REGION Network 13: CALL FB31 SPINDLE C24
   // 2#0000_0001 OPTIONS 0 BIT 0 MEASURING SYSTEM 2 OPTION
   // 2#0000_0010 OPTIONS 0 BIT 1 BELT BROKEN OPTION
   // 2#0000_0100 OPTIONS 0 BIT 2 COOLING OPTION
   // 2#0000_1000 OPTIONS 0 BIT 3 MQL OR HP OPTION
   // 2#0001_0000 OPTIONS 0 BIT 4 ANALOG TEMPERATURE SENSOR OPTION
   // 2#0010_0000 OPTIONS 0 BIT 5 PTC TEMPERATURE SENSOR OPTION
   // 2#0100_0000 OPTIONS 0 BIT 6 TWIN KESSLER VPM READY OPTION
   // 2#1000_0000 OPTIONS 0 BIT 7 MPP SPINDLE OVERRIDE OPTION
   // 
   // 2#0000_0001 OPTIONS 1 BIT 0 SPARE OPTION
   // 2#0000_0010 OPTIONS 1 BIT 1 SPARE OPTION
   // 2#0000_0100 OPTIONS 1 BIT 2 SPARE OPTION
   // 2#0000_1000 OPTIONS 1 BIT 3 SPARE OPTION
   // 2#0001_0000 OPTIONS 1 BIT 4 SPARE OPTION
   // 2#0010_0000 OPTIONS 1 BIT 5 SPARE OPTION
   // 2#0100_0000 OPTIONS 1 BIT 6 SPARE OPTION
   // 2#1000_0000 OPTIONS 1 BIT 7 SPARE OPTION
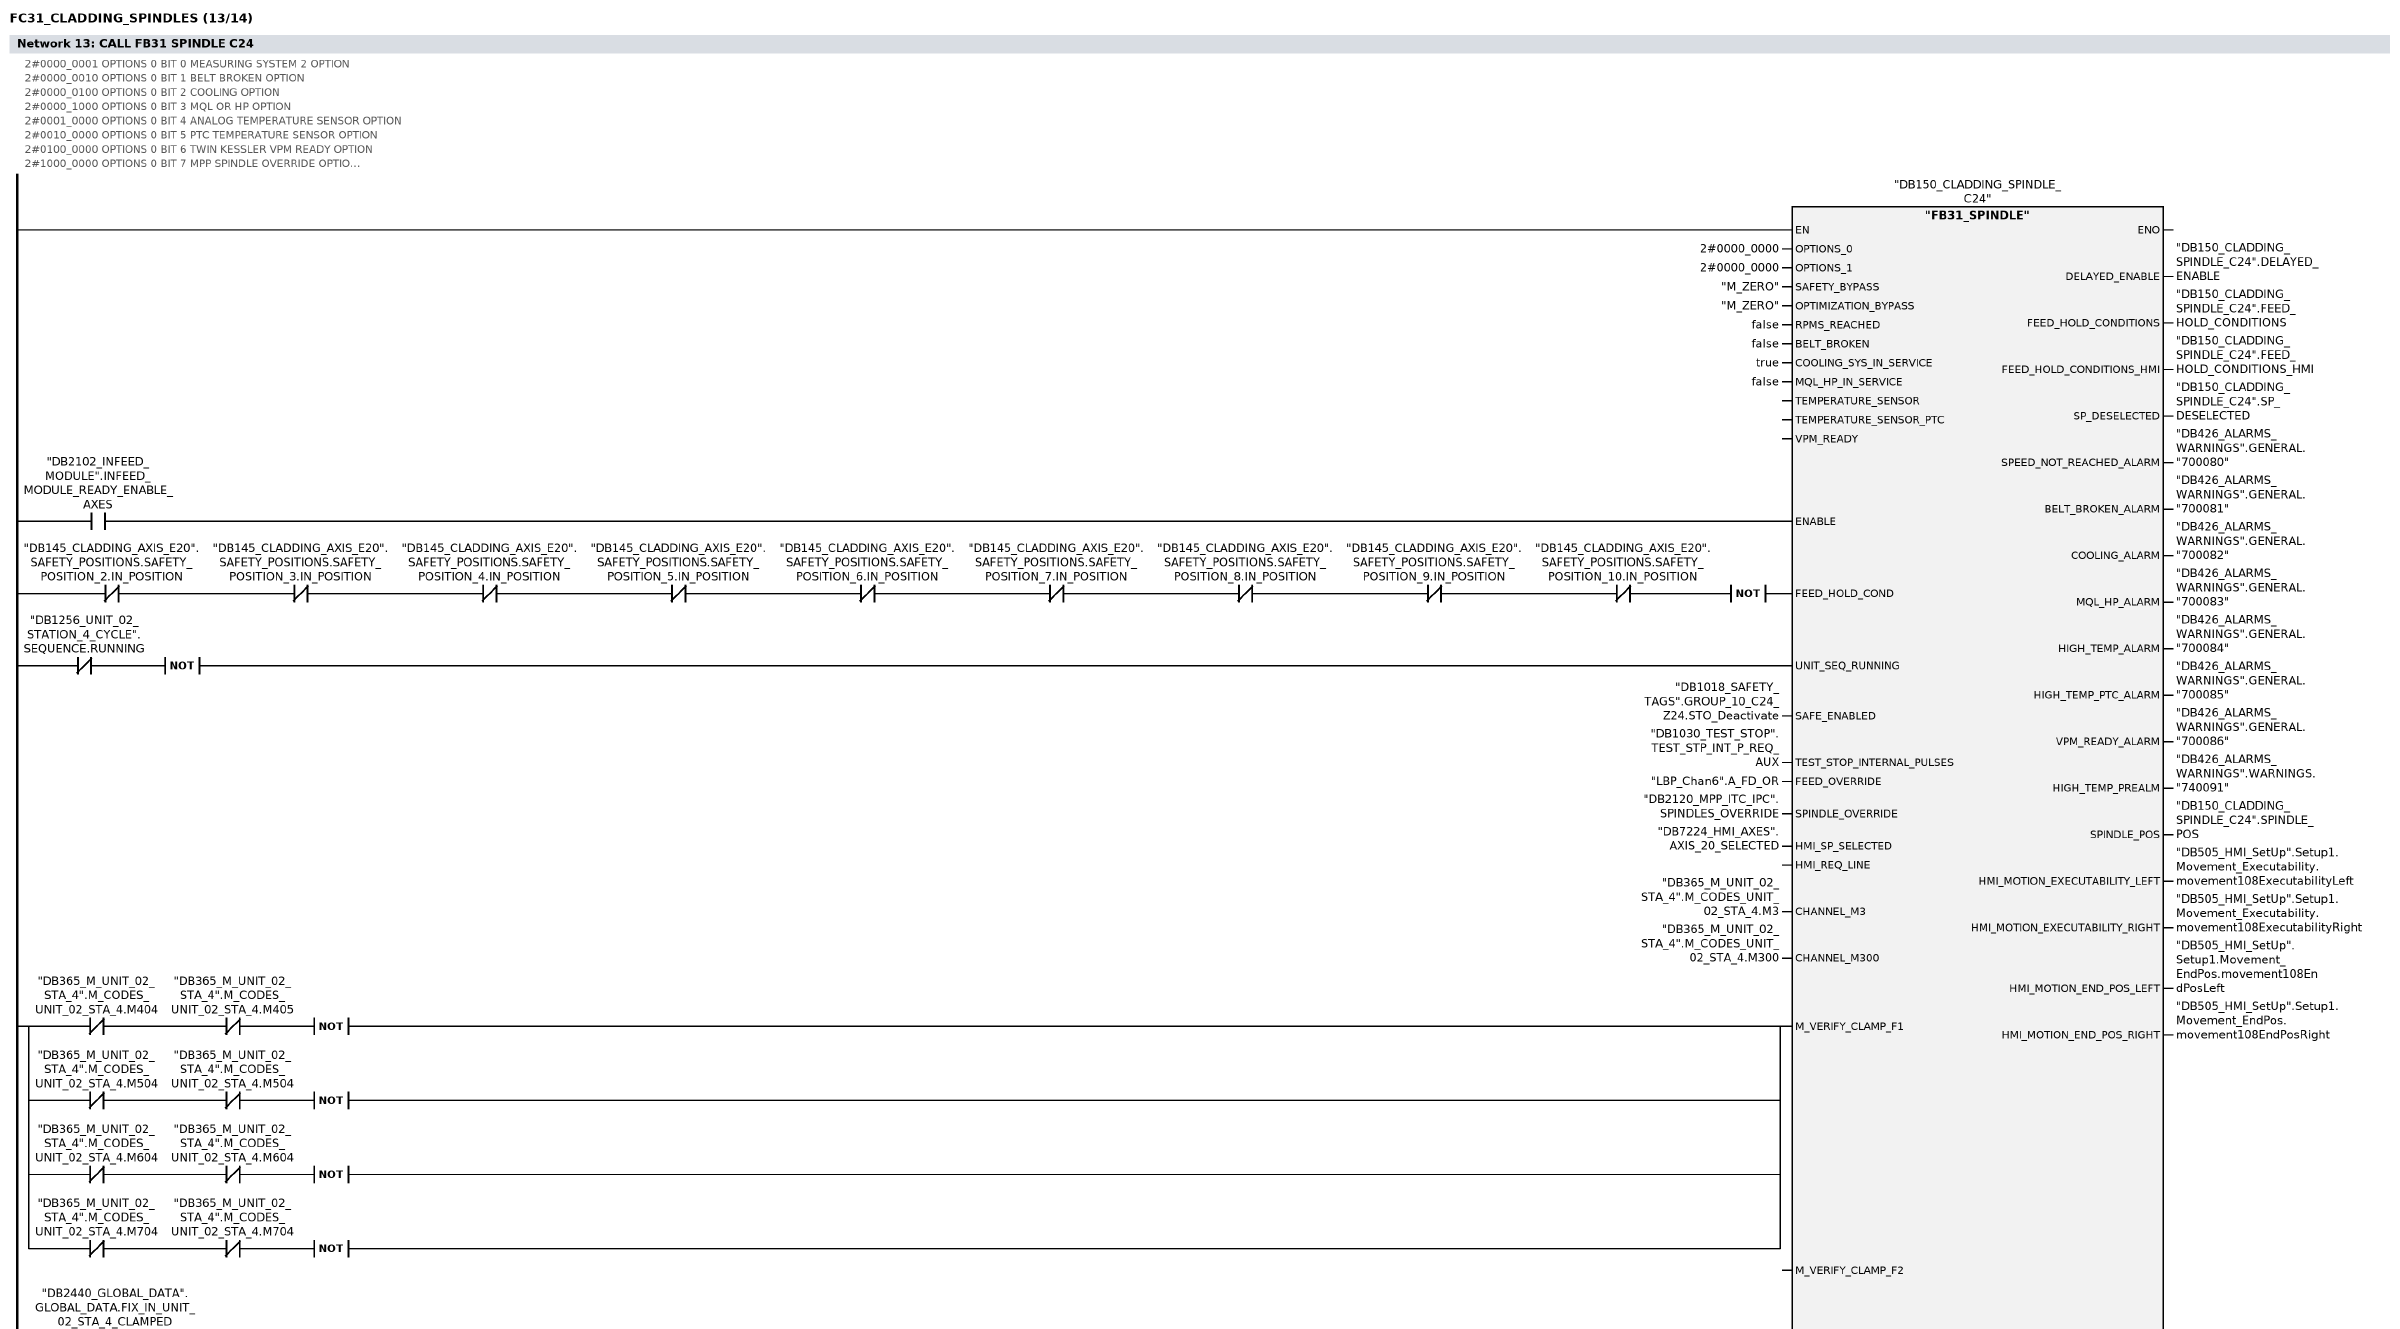
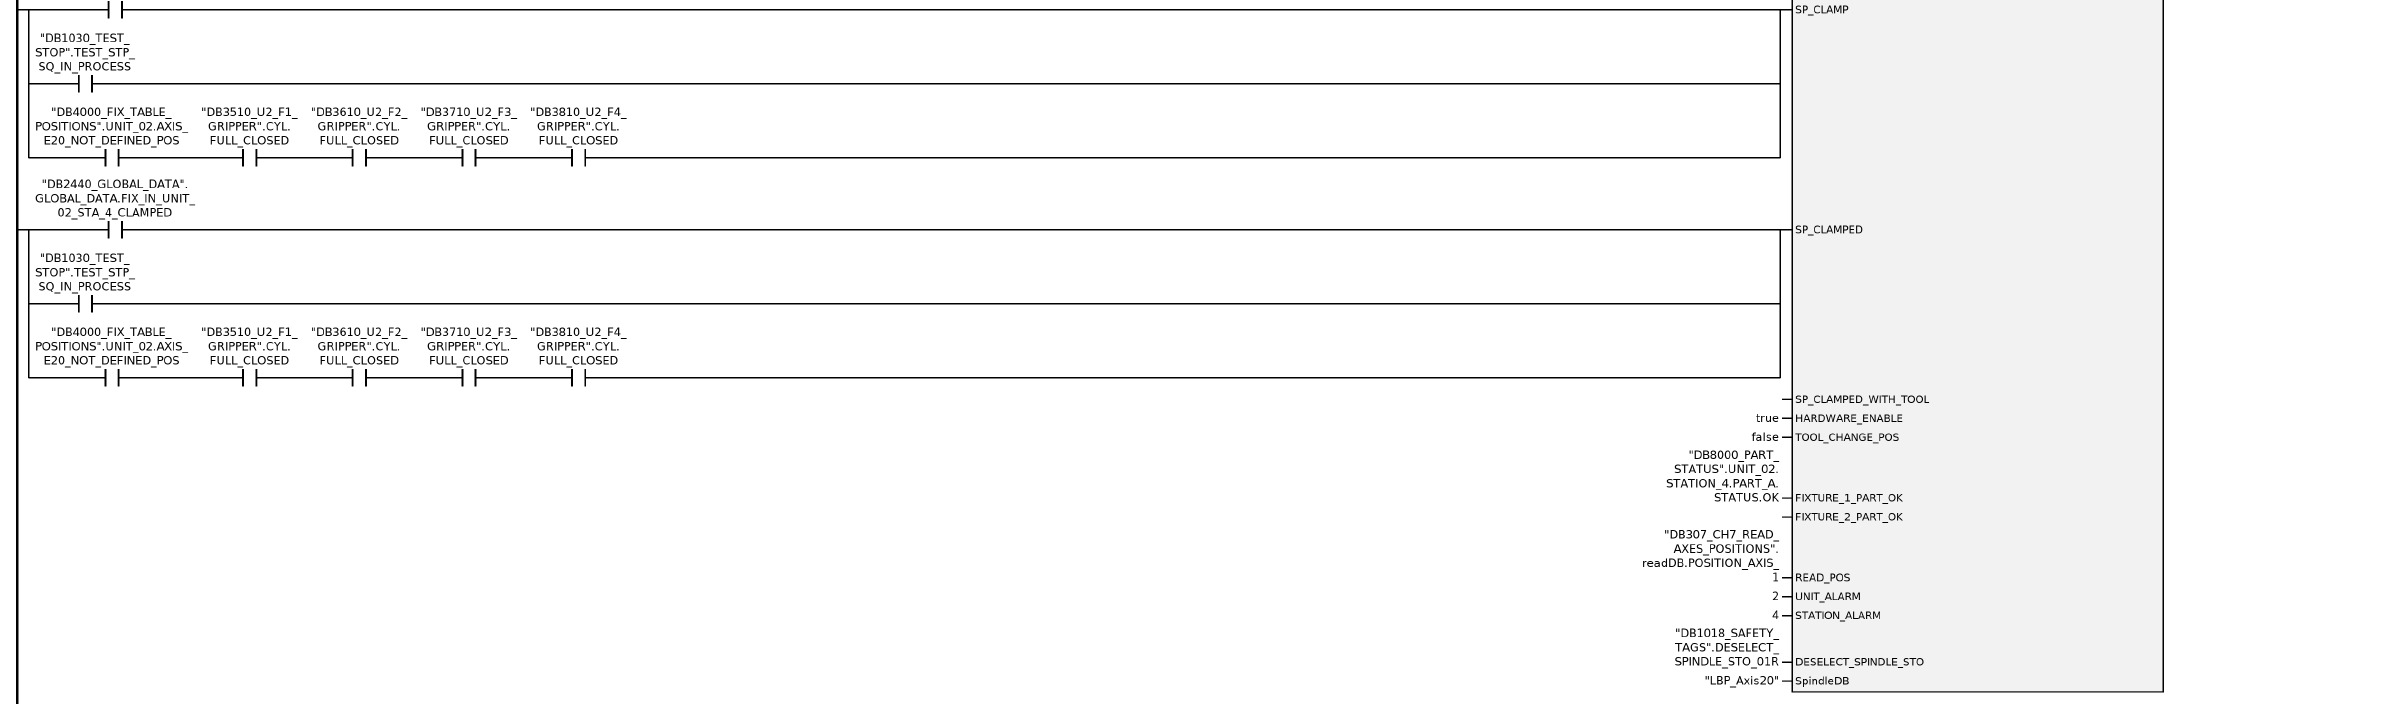
   RUNG wire#powerrail
      "DB150_CLADDING_SPINDLE_C24"(ENABLE := wire#w1, FEED_HOLD_COND := wire#w2, UNIT_SEQ_RUNNING := wire#w3, M_VERIFY_CLAMP_F1 := wire#w4, SP_CLAMP := wire#w5, SP_CLAMPED := wire#w6, OPTIONS_0 := 2#0000_0000, OPTIONS_1 := 2#0000_0000, SAFETY_BYPASS := "M_ZERO", OPTIMIZATION_BYPASS := "M_ZERO", RPMS_REACHED := false, BELT_BROKEN := false, COOLING_SYS_IN_SERVICE := true, MQL_HP_IN_SERVICE := false, TEMPERATURE_SENSOR :=, TEMPERATURE_SENSOR_PTC :=, VPM_READY :=, SAFE_ENABLED := "DB1018_SAFETY_TAGS".GROUP_10_C24_Z24.STO_Deactivate, TEST_STOP_INTERNAL_PULSES := "DB1030_TEST_STOP".TEST_STP_INT_P_REQ_AUX, FEED_OVERRIDE := "LBP_Chan6".A_FD_OR, SPINDLE_OVERRIDE := "DB2120_MPP_ITC_IPC".SPINDLES_OVERRIDE, HMI_SP_SELECTED := "DB7224_HMI_AXES".AXIS_20_SELECTED, HMI_REQ_LINE :=, CHANNEL_M3 := "DB365_M_UNIT_02_STA_4".M_CODES_UNIT_02_STA_4.M3, CHANNEL_M300 := "DB365_M_UNIT_02_STA_4".M_CODES_UNIT_02_STA_4.M300, M_VERIFY_CLAMP_F2 :=, SP_CLAMPED_WITH_TOOL :=, HARDWARE_ENABLE := true, TOOL_CHANGE_POS := false, FIXTURE_1_PART_OK := "DB8000_PART_STATUS".UNIT_02.STATION_4.PART_A.STATUS.OK, FIXTURE_2_PART_OK :=, READ_POS := "DB307_CH7_READ_AXES_POSITIONS".readDB.POSITION_AXIS_1, UNIT_ALARM := 2, STATION_ALARM := 4, DESELECT_SPINDLE_STO := "DB1018_SAFETY_TAGS".DESELECT_SPINDLE_STO_01R, SpindleDB := "LBP_Axis20", DELAYED_ENABLE => "DB150_CLADDING_SPINDLE_C24".DELAYED_ENABLE, FEED_HOLD_CONDITIONS => "DB150_CLADDING_SPINDLE_C24".FEED_HOLD_CONDITIONS, FEED_HOLD_CONDITIONS_HMI => "DB150_CLADDING_SPINDLE_C24".FEED_HOLD_CONDITIONS_HMI, SP_DESELECTED => "DB150_CLADDING_SPINDLE_C24".SP_DESELECTED, SPEED_NOT_REACHED_ALARM => "DB426_ALARMS_WARNINGS".GENERAL."700080", BELT_BROKEN_ALARM => "DB426_ALARMS_WARNINGS".GENERAL."700081", COOLING_ALARM => "DB426_ALARMS_WARNINGS".GENERAL."700082", MQL_HP_ALARM => "DB426_ALARMS_WARNINGS".GENERAL."700083", HIGH_TEMP_ALARM => "DB426_ALARMS_WARNINGS".GENERAL."700084", HIGH_TEMP_PTC_ALARM => "DB426_ALARMS_WARNINGS".GENERAL."700085", VPM_READY_ALARM => "DB426_ALARMS_WARNINGS".GENERAL."700086", HIGH_TEMP_PREALM => "DB426_ALARMS_WARNINGS".WARNINGS."740091", SPINDLE_POS => "DB150_CLADDING_SPINDLE_C24".SPINDLE_POS, HMI_MOTION_EXECUTABILITY_LEFT => "DB505_HMI_SetUp".Setup1.Movement_Executability.movement108ExecutabilityLeft, HMI_MOTION_EXECUTABILITY_RIGHT => "DB505_HMI_SetUp".Setup1.Movement_Executability.movement108ExecutabilityRight, HMI_MOTION_END_POS_LEFT => "DB505_HMI_SetUp".Setup1.Movement_EndPos.movement108EndPosLeft, HMI_MOTION_END_POS_RIGHT => "DB505_HMI_SetUp".Setup1.Movement_EndPos.movement108EndPosRight)
   END_RUNG
   RUNG wire#powerrail
      Contact( "DB2102_INFEED_MODULE".INFEED_MODULE_READY_ENABLE_AXES )
   END_RUNG wire#w1
   RUNG wire#powerrail
      I_Contact( "DB145_CLADDING_AXIS_E20".SAFETY_POSITIONS.SAFETY_POSITION_2.IN_POSITION )
      I_Contact( "DB145_CLADDING_AXIS_E20".SAFETY_POSITIONS.SAFETY_POSITION_3.IN_POSITION )
      I_Contact( "DB145_CLADDING_AXIS_E20".SAFETY_POSITIONS.SAFETY_POSITION_4.IN_POSITION )
      I_Contact( "DB145_CLADDING_AXIS_E20".SAFETY_POSITIONS.SAFETY_POSITION_5.IN_POSITION )
      I_Contact( "DB145_CLADDING_AXIS_E20".SAFETY_POSITIONS.SAFETY_POSITION_6.IN_POSITION )
      I_Contact( "DB145_CLADDING_AXIS_E20".SAFETY_POSITIONS.SAFETY_POSITION_7.IN_POSITION )
      I_Contact( "DB145_CLADDING_AXIS_E20".SAFETY_POSITIONS.SAFETY_POSITION_8.IN_POSITION )
      I_Contact( "DB145_CLADDING_AXIS_E20".SAFETY_POSITIONS.SAFETY_POSITION_9.IN_POSITION )
      I_Contact( "DB145_CLADDING_AXIS_E20".SAFETY_POSITIONS.SAFETY_POSITION_10.IN_POSITION )
      Not()
   END_RUNG wire#w2
   RUNG wire#powerrail
      I_Contact( "DB1256_UNIT_02_STATION_4_CYCLE".SEQUENCE.RUNNING )
      Not()
   END_RUNG wire#w3
   RUNG wire#powerrail
      I_Contact( "DB365_M_UNIT_02_STA_4".M_CODES_UNIT_02_STA_4.M404 )
      I_Contact( "DB365_M_UNIT_02_STA_4".M_CODES_UNIT_02_STA_4.M405 )
      Not()
   END_RUNG wire#w4
   RUNG wire#powerrail
      I_Contact( "DB365_M_UNIT_02_STA_4".M_CODES_UNIT_02_STA_4.M504 )
      I_Contact( "DB365_M_UNIT_02_STA_4".M_CODES_UNIT_02_STA_4.M504 )
      Not()
   END_RUNG wire#w4
   RUNG wire#powerrail
      I_Contact( "DB365_M_UNIT_02_STA_4".M_CODES_UNIT_02_STA_4.M604 )
      I_Contact( "DB365_M_UNIT_02_STA_4".M_CODES_UNIT_02_STA_4.M604 )
      Not()
   END_RUNG wire#w4
   RUNG wire#powerrail
      I_Contact( "DB365_M_UNIT_02_STA_4".M_CODES_UNIT_02_STA_4.M704 )
      I_Contact( "DB365_M_UNIT_02_STA_4".M_CODES_UNIT_02_STA_4.M704 )
      Not()
   END_RUNG wire#w4
   RUNG wire#powerrail
      Contact( "DB2440_GLOBAL_DATA".GLOBAL_DATA.FIX_IN_UNIT_02_STA_4_CLAMPED )
   END_RUNG wire#w5
   RUNG wire#powerrail
      Contact( "DB1030_TEST_STOP".TEST_STP_SQ_IN_PROCESS )
   END_RUNG wire#w5
   RUNG wire#powerrail
      Contact( "DB4000_FIX_TABLE_POSITIONS".UNIT_02.AXIS_E20_NOT_DEFINED_POS )
      Contact( "DB3510_U2_F1_GRIPPER".CYL.FULL_CLOSED )
      Contact( "DB3610_U2_F2_GRIPPER".CYL.FULL_CLOSED )
      Contact( "DB3710_U2_F3_GRIPPER".CYL.FULL_CLOSED )
      Contact( "DB3810_U2_F4_GRIPPER".CYL.FULL_CLOSED )
   END_RUNG wire#w5
   RUNG wire#powerrail
      Contact( "DB2440_GLOBAL_DATA".GLOBAL_DATA.FIX_IN_UNIT_02_STA_4_CLAMPED )
   END_RUNG wire#w6
   RUNG wire#powerrail
      Contact( "DB1030_TEST_STOP".TEST_STP_SQ_IN_PROCESS )
   END_RUNG wire#w6
   RUNG wire#powerrail
      Contact( "DB4000_FIX_TABLE_POSITIONS".UNIT_02.AXIS_E20_NOT_DEFINED_POS )
      Contact( "DB3510_U2_F1_GRIPPER".CYL.FULL_CLOSED )
      Contact( "DB3610_U2_F2_GRIPPER".CYL.FULL_CLOSED )
      Contact( "DB3710_U2_F3_GRIPPER".CYL.FULL_CLOSED )
      Contact( "DB3810_U2_F4_GRIPPER".CYL.FULL_CLOSED )
   END_RUNG wire#w6
   // the same network as SCL:
   "DB150_CLADDING_SPINDLE_C24"(OPTIONS_0 := 2#0000_0000,   // "FB31_SPINDLE"
                           OPTIONS_1 := 2#0000_0000,
                           SAFETY_BYPASS := "M_ZERO",
                           OPTIMIZATION_BYPASS := "M_ZERO",
                           RPMS_REACHED := false,
                           BELT_BROKEN := false,
                           COOLING_SYS_IN_SERVICE := true,
                           MQL_HP_IN_SERVICE := false,
                           ENABLE := "DB2102_INFEED_MODULE".INFEED_MODULE_READY_ENABLE_AXES,
                           FEED_HOLD_COND := NOT (NOT "DB145_CLADDING_AXIS_E20".SAFETY_POSITIONS.SAFETY_POSITION_2.IN_POSITION AND NOT "DB145_CLADDING_AXIS_E20".SAFETY_POSITIONS.SAFETY_POSITION_3.IN_POSITION AND NOT "DB145_CLADDING_AXIS_E20".SAFETY_POSITIONS.SAFETY_POSITION_4.IN_POSITION AND NOT "DB145_CLADDING_AXIS_E20".SAFETY_POSITIONS.SAFETY_POSITION_5.IN_POSITION AND NOT "DB145_CLADDING_AXIS_E20".SAFETY_POSITIONS.SAFETY_POSITION_6.IN_POSITION AND NOT "DB145_CLADDING_AXIS_E20".SAFETY_POSITIONS.SAFETY_POSITION_7.IN_POSITION AND NOT "DB145_CLADDING_AXIS_E20".SAFETY_POSITIONS.SAFETY_POSITION_8.IN_POSITION AND NOT "DB145_CLADDING_AXIS_E20".SAFETY_POSITIONS.SAFETY_POSITION_9.IN_POSITION AND NOT "DB145_CLADDING_AXIS_E20".SAFETY_POSITIONS.SAFETY_POSITION_10.IN_POSITION),
                           UNIT_SEQ_RUNNING := NOT (NOT "DB1256_UNIT_02_STATION_4_CYCLE".SEQUENCE.RUNNING),
                           SAFE_ENABLED := "DB1018_SAFETY_TAGS".GROUP_10_C24_Z24.STO_Deactivate,
                           TEST_STOP_INTERNAL_PULSES := "DB1030_TEST_STOP".TEST_STP_INT_P_REQ_AUX,
                           FEED_OVERRIDE := "LBP_Chan6".A_FD_OR,
                           SPINDLE_OVERRIDE := "DB2120_MPP_ITC_IPC".SPINDLES_OVERRIDE,
                           HMI_SP_SELECTED := "DB7224_HMI_AXES".AXIS_20_SELECTED,
                           CHANNEL_M3 := "DB365_M_UNIT_02_STA_4".M_CODES_UNIT_02_STA_4.M3,
                           CHANNEL_M300 := "DB365_M_UNIT_02_STA_4".M_CODES_UNIT_02_STA_4.M300,
                           M_VERIFY_CLAMP_F1 := NOT (NOT "DB365_M_UNIT_02_STA_4".M_CODES_UNIT_02_STA_4.M404 AND NOT "DB365_M_UNIT_02_STA_4".M_CODES_UNIT_02_STA_4.M405) OR NOT (NOT "DB365_M_UNIT_02_STA_4".M_CODES_UNIT_02_STA_4.M504 AND NOT "DB365_M_UNIT_02_STA_4".M_CODES_UNIT_02_STA_4.M504) OR NOT (NOT "DB365_M_UNIT_02_STA_4".M_CODES_UNIT_02_STA_4.M604 AND NOT "DB365_M_UNIT_02_STA_4".M_CODES_UNIT_02_STA_4.M604) OR NOT (NOT "DB365_M_UNIT_02_STA_4".M_CODES_UNIT_02_STA_4.M704 AND NOT "DB365_M_UNIT_02_STA_4".M_CODES_UNIT_02_STA_4.M704),
                           SP_CLAMP := "DB2440_GLOBAL_DATA".GLOBAL_DATA.FIX_IN_UNIT_02_STA_4_CLAMPED OR "DB1030_TEST_STOP".TEST_STP_SQ_IN_PROCESS OR ("DB4000_FIX_TABLE_POSITIONS".UNIT_02.AXIS_E20_NOT_DEFINED_POS AND "DB3510_U2_F1_GRIPPER".CYL.FULL_CLOSED AND "DB3610_U2_F2_GRIPPER".CYL.FULL_CLOSED AND "DB3710_U2_F3_GRIPPER".CYL.FULL_CLOSED AND "DB3810_U2_F4_GRIPPER".CYL.FULL_CLOSED),
                           SP_CLAMPED := "DB2440_GLOBAL_DATA".GLOBAL_DATA.FIX_IN_UNIT_02_STA_4_CLAMPED OR "DB1030_TEST_STOP".TEST_STP_SQ_IN_PROCESS OR ("DB4000_FIX_TABLE_POSITIONS".UNIT_02.AXIS_E20_NOT_DEFINED_POS AND "DB3510_U2_F1_GRIPPER".CYL.FULL_CLOSED AND "DB3610_U2_F2_GRIPPER".CYL.FULL_CLOSED AND "DB3710_U2_F3_GRIPPER".CYL.FULL_CLOSED AND "DB3810_U2_F4_GRIPPER".CYL.FULL_CLOSED),
                           HARDWARE_ENABLE := true,
                           TOOL_CHANGE_POS := false,
                           FIXTURE_1_PART_OK := "DB8000_PART_STATUS".UNIT_02.STATION_4.PART_A.STATUS.OK,
                           READ_POS := "DB307_CH7_READ_AXES_POSITIONS".readDB.POSITION_AXIS_1,
                           UNIT_ALARM := 2,
                           STATION_ALARM := 4,
                           DESELECT_SPINDLE_STO := "DB1018_SAFETY_TAGS".DESELECT_SPINDLE_STO_01R,
                           SpindleDB := "LBP_Axis20",
                           DELAYED_ENABLE => "DB150_CLADDING_SPINDLE_C24".DELAYED_ENABLE,
                           FEED_HOLD_CONDITIONS => "DB150_CLADDING_SPINDLE_C24".FEED_HOLD_CONDITIONS,
                           FEED_HOLD_CONDITIONS_HMI => "DB150_CLADDING_SPINDLE_C24".FEED_HOLD_CONDITIONS_HMI,
                           SP_DESELECTED => "DB150_CLADDING_SPINDLE_C24".SP_DESELECTED,
                           SPEED_NOT_REACHED_ALARM => "DB426_ALARMS_WARNINGS".GENERAL."700080",
                           BELT_BROKEN_ALARM => "DB426_ALARMS_WARNINGS".GENERAL."700081",
                           COOLING_ALARM => "DB426_ALARMS_WARNINGS".GENERAL."700082",
                           MQL_HP_ALARM => "DB426_ALARMS_WARNINGS".GENERAL."700083",
                           HIGH_TEMP_ALARM => "DB426_ALARMS_WARNINGS".GENERAL."700084",
                           HIGH_TEMP_PTC_ALARM => "DB426_ALARMS_WARNINGS".GENERAL."700085",
                           VPM_READY_ALARM => "DB426_ALARMS_WARNINGS".GENERAL."700086",
                           HIGH_TEMP_PREALM => "DB426_ALARMS_WARNINGS".WARNINGS."740091",
                           SPINDLE_POS => "DB150_CLADDING_SPINDLE_C24".SPINDLE_POS,
                           HMI_MOTION_EXECUTABILITY_LEFT => "DB505_HMI_SetUp".Setup1.Movement_Executability.movement108ExecutabilityLeft,
                           HMI_MOTION_EXECUTABILITY_RIGHT => "DB505_HMI_SetUp".Setup1.Movement_Executability.movement108ExecutabilityRight,
                           HMI_MOTION_END_POS_LEFT => "DB505_HMI_SetUp".Setup1.Movement_EndPos.movement108EndPosLeft,
                           HMI_MOTION_END_POS_RIGHT => "DB505_HMI_SetUp".Setup1.Movement_EndPos.movement108EndPosRight);
END_REGION

REGION Network 14: SPINDLE C24 OPERATOR HELP
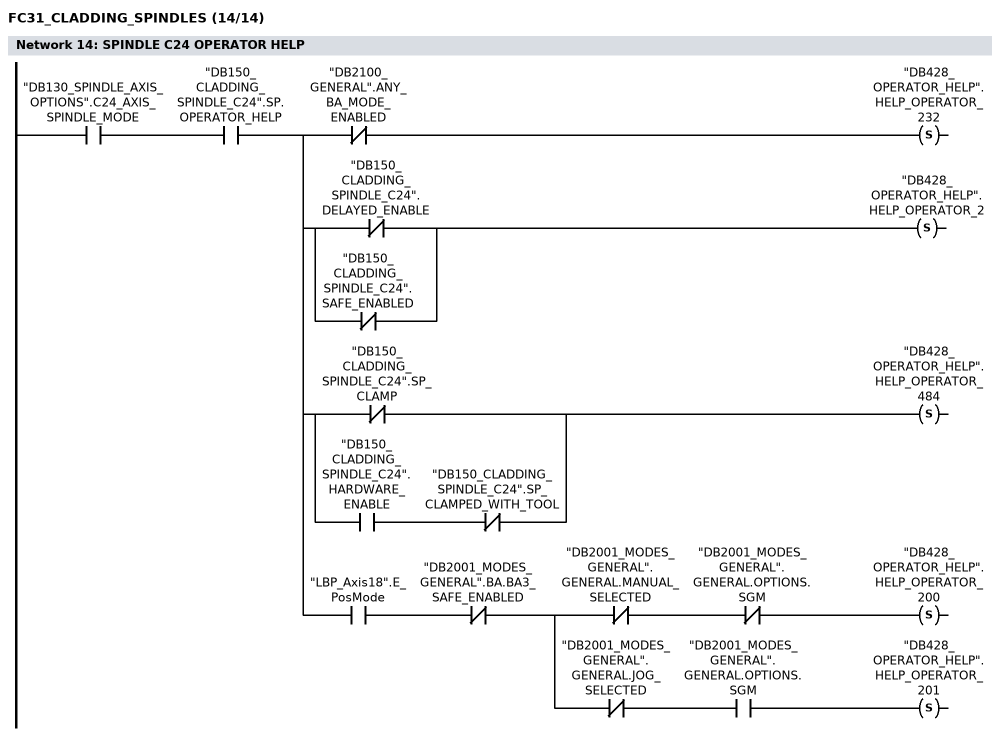
   RUNG wire#powerrail
      Contact( "DB130_SPINDLE_AXIS_OPTIONS".C24_AXIS_SPINDLE_MODE )
      Contact( "DB150_CLADDING_SPINDLE_C24".SP.OPERATOR_HELP )
      wire#w1
      I_Contact( "DB2100_GENERAL".ANY_BA_MODE_ENABLED )
      S_Coil( "DB428_OPERATOR_HELP".HELP_OPERATOR_232 )
   END_RUNG
   RUNG wire#w1
      I_Contact( "DB150_CLADDING_SPINDLE_C24".DELAYED_ENABLE )
      wire#w2
      S_Coil( "DB428_OPERATOR_HELP".HELP_OPERATOR_2 )
   END_RUNG
   RUNG wire#w1
      I_Contact( "DB150_CLADDING_SPINDLE_C24".SAFE_ENABLED )
   END_RUNG wire#w2
   RUNG wire#w1
      I_Contact( "DB150_CLADDING_SPINDLE_C24".SP_CLAMP )
      wire#w3
      S_Coil( "DB428_OPERATOR_HELP".HELP_OPERATOR_484 )
   END_RUNG
   RUNG wire#w1
      Contact( "DB150_CLADDING_SPINDLE_C24".HARDWARE_ENABLE )
      I_Contact( "DB150_CLADDING_SPINDLE_C24".SP_CLAMPED_WITH_TOOL )
   END_RUNG wire#w3
   RUNG wire#w1
      Contact( "LBP_Axis18".E_PosMode )
      I_Contact( "DB2001_MODES_GENERAL".BA.BA3_SAFE_ENABLED )
      wire#w4
      I_Contact( "DB2001_MODES_GENERAL".GENERAL.MANUAL_SELECTED )
      I_Contact( "DB2001_MODES_GENERAL".GENERAL.OPTIONS.SGM )
      S_Coil( "DB428_OPERATOR_HELP".HELP_OPERATOR_200 )
   END_RUNG
   RUNG wire#w4
      I_Contact( "DB2001_MODES_GENERAL".GENERAL.JOG_SELECTED )
      Contact( "DB2001_MODES_GENERAL".GENERAL.OPTIONS.SGM )
      S_Coil( "DB428_OPERATOR_HELP".HELP_OPERATOR_201 )
   END_RUNG
   // the same network as SCL:
   #_w1 := "DB130_SPINDLE_AXIS_OPTIONS".C24_AXIS_SPINDLE_MODE AND "DB150_CLADDING_SPINDLE_C24".SP.OPERATOR_HELP;
   IF #_w1 AND NOT "DB2100_GENERAL".ANY_BA_MODE_ENABLED THEN
       "DB428_OPERATOR_HELP".HELP_OPERATOR_232 := TRUE;
   END_IF;
   IF #_w1 AND (NOT "DB150_CLADDING_SPINDLE_C24".DELAYED_ENABLE OR NOT "DB150_CLADDING_SPINDLE_C24".SAFE_ENABLED) THEN
       "DB428_OPERATOR_HELP".HELP_OPERATOR_2 := TRUE;
   END_IF;
   IF #_w1 AND (NOT "DB150_CLADDING_SPINDLE_C24".SP_CLAMP OR ("DB150_CLADDING_SPINDLE_C24".HARDWARE_ENABLE AND NOT "DB150_CLADDING_SPINDLE_C24".SP_CLAMPED_WITH_TOOL)) THEN
       "DB428_OPERATOR_HELP".HELP_OPERATOR_484 := TRUE;
   END_IF;
   #_w2 := #_w1 AND "LBP_Axis18".E_PosMode AND NOT "DB2001_MODES_GENERAL".BA.BA3_SAFE_ENABLED;
   IF #_w2 AND NOT "DB2001_MODES_GENERAL".GENERAL.MANUAL_SELECTED AND NOT "DB2001_MODES_GENERAL".GENERAL.OPTIONS.SGM THEN
       "DB428_OPERATOR_HELP".HELP_OPERATOR_200 := TRUE;
   END_IF;
   IF #_w2 AND NOT "DB2001_MODES_GENERAL".GENERAL.JOG_SELECTED AND "DB2001_MODES_GENERAL".GENERAL.OPTIONS.SGM THEN
       "DB428_OPERATOR_HELP".HELP_OPERATOR_201 := TRUE;
   END_IF;
END_REGION
END_FUNCTION
